(* CODESYS project 1210_xlh_terminal_manager.project
   Description: Receives some incoming messages and echoes them with CAN-ID +1
   Company: 3S - Smart Software Solutions GmbH
   Version: 1.0.0.0
   Title: CAN Bus API Example
   Author: 3S - Smart Software Solutions GmbH

Project tree, tasks and I/O mapping:
  xLH_base : CODESYS Control for Raspberry Pi 64 SL, CODESYS, order no. 2302000009, version 4.20.0.0
    application app
      libraries: Standard, 3.5.22.0 (System); Util, 3.5.22.0 (System); VisuDialogs, * (System); Memory, * (3S - Smart Software Solutions GmbH); CmpBitmapPool, * (System); CAN API, 1.0.0.4 (CODESYS); MemoryUtils, * (3S - Smart Software Solutions GmbH); CAA CiA 405, 4.3.0.0 (CODESYS)
      task CAN_OPEN_TASK (cyclic, interval 1 ms, priority 0) calls nothing
      task VISU_TASK (cyclic, interval 100 ms, priority 31) calls VisuElems.Visu_Prg
      task MAIN_TASK (cyclic, interval 4 ms, priority 1) calls MAIN_CALLER
      program MAIN_CALLER [ST]
      function block FB_SDO_READ_4_BYTE [ST]
      visualisation Visualization
      trace Trace (task MAIN_TASK): MAIN.diPosition, MAIN.iSetSpeed, MAIN.iDebug2Pos, MAIN.iDebug1Mileage, MAIN.auiUltrasonic[1], MAIN.fbReadStatusLoopTime.udiValue, MAIN.iSpeed2, MAIN.iSpeed1, MAIN.iPitch
      data type MOTION_CONTROL_BYTE
      program MAIN [ST]
      function block FB_XLH_TERMINAL [ST]: read, write
      TOOLBOX/
        GPIO/
          function block FB_XLH_GPIO [CFC]
          function block FB_XLH_SWITCH_BUTTON_LED [CFC]
        data type RGB
        data type UNION_BYTE_INT
      program io [ST]
    CANbus : CANbus, CODESYS, version 4.3.0.0
        settings: Baudrate = 1000 kbit/s
      CANopen_Manager : CANopen_Manager, CODESYS, version 4.3.0.0
          settings: NMT Start All = TRUE; Polling of optional slaves = FALSE; ConfigVersion = 50659584
        xlh_terminal : xlh_terminal, xemax ag, order no. 0, version Revision=16#00000001, FileVersion=1.0
            settings: NODEIDSAVED = 3; SDO Timeout = 1000000; PDO_Autoconfig = FALSE; EXPERTSETTINGS = FALSE; PDO 16#1400.COBID = 16#00000203; Process by CANopenManager = TRUE; PDO 16#1401.COBID = 16#00000303; Process by CANopenManager = TRUE; PDO 16#1402.COBID = 16#00000403; Process by CANopenManager = TRUE; PDO 16#1403.COBID = 16#00000503; Process by CANopenManager = TRUE; PDO 16#1800.COBID = 16#00000183; Process by CANopenManager = TRUE; PDO 16#1801.COBID = 16#00000283; Process by CANopenManager = TRUE; PDO 16#1802.COBID = 16#00000383; Process by CANopenManager = TRUE; PDO 16#1803.COBID = 16#00000483; Process by CANopenManager = TRUE; Data out 1 Byte 0.Subindex = 16#01; Data out 1 Byte 1.Subindex = 16#02; Data out 1 Byte 2.Subindex = 16#03; Data out 1 Byte 3.Subindex = 16#04; Data out 1 Byte 4.Subindex = 16#05; Data out 1 Byte 5.Subindex = 16#06; Data out 1 Byte 6.Subindex = 16#07; Data out 1 Byte 7.Subindex = 16#08; Data out 2 Byte 0.Subindex = 16#01; Data out 2 Byte 1.Subindex = 16#02; Data out 2 Byte 2.Subindex = 16#03; Data out 2 Byte 3.Subindex = 16#04; Data out 2 Byte 4.Subindex = 16#05; Data out 2 Byte 5.Subindex = 16#06; Data out 2 Byte 6.Subindex = 16#07; Data out 2 Byte 7.Subindex = 16#08; Data out 3 Byte 0.Subindex = 16#01; Data out 3 Byte 1.Subindex = 16#02; Data out 3 Byte 2.Subindex = 16#03; Data out 3 Byte 3.Subindex = 16#04;
              Data out 3 Byte 4.Subindex = 16#05; Data out 3 Byte 5.Subindex = 16#06; Data out 3 Byte 6.Subindex = 16#07; Data out 3 Byte 7.Subindex = 16#08; Data out 4 Byte 0.Subindex = 16#01; Data out 4 Byte 1.Subindex = 16#02; Data out 4 Byte 2.Subindex = 16#03; Data out 4 Byte 3.Subindex = 16#04; Data out 4 Byte 4.Subindex = 16#05; Data out 4 Byte 5.Subindex = 16#06; Data out 4 Byte 6.Subindex = 16#07; Data out 4 Byte 7.Subindex = 16#08; Data in 1 Byte 0.Subindex = 16#01; Data in 1 Byte 1.Subindex = 16#02; Data in 1 Byte 2.Subindex = 16#03; Data in 1 Byte 3.Subindex = 16#04; Data in 1 Byte 4.Subindex = 16#05; Data in 1 Byte 5.Subindex = 16#06; Data in 1 Byte 6.Subindex = 16#07; Data in 1 Byte 7.Subindex = 16#08; Data in 2 Byte 0.Subindex = 16#01; Data in 2 Byte 1.Subindex = 16#02; Data in 2 Byte 2.Subindex = 16#03; Data in 2 Byte 3.Subindex = 16#04; Data in 2 Byte 4.Subindex = 16#05; Data in 2 Byte 5.Subindex = 16#06; Data in 2 Byte 6.Subindex = 16#07; Data in 2 Byte 7.Subindex = 16#08; Data in 3 Byte 0.Subindex = 16#01; Data in 3 Byte 1.Subindex = 16#02; Data in 3 Byte 2.Subindex = 16#03; Data in 3 Byte 3.Subindex = 16#04; Data in 3 Byte 4.Subindex = 16#05; Data in 3 Byte 5.Subindex = 16#06; Data in 3 Byte 6.Subindex = 16#07; Data in 3 Byte 7.Subindex = 16#08; Data in 4 Byte 0.Subindex = 16#01; Data in 4 Byte 1.Subindex = 16#02; Data in 4 Byte 2.Subindex = 16#03; Data in 4 Byte 3.Subindex = 16#04;
              Data in 4 Byte 4.Subindex = 16#05; Data in 4 Byte 5.Subindex = 16#06; Data in 4 Byte 6.Subindex = 16#07; Data in 4 Byte 7.Subindex = 16#08; SDO List.Set COB-ID sync.Index = 16#1005; SDO List.Set COB-ID sync.Subindex = 16#00; SDO List.Set COB-ID sync.Value = 16#00000080; SDO List.Set COB-ID sync.Size = 32; SDO List.Set COB-ID sync.AbortIfError = FALSE; SDO List.Set COB-ID sync.JumpToLine = FALSE; SDO List.Set COB-ID sync.Line = 0; SDO List.Set communication cycle period.Index = 16#1006; SDO List.Set communication cycle period.Subindex = 16#00; SDO List.Set communication cycle period.Value = 16#00000000; SDO List.Set communication cycle period.Size = 32; SDO List.Set communication cycle period.AbortIfError = FALSE; SDO List.Set communication cycle period.JumpToLine = FALSE; SDO List.Set communication cycle period.Line = 0; SDO List.Set Guardtime.Index = 16#100C; SDO List.Set Guardtime.Subindex = 16#00; SDO List.Set Guardtime.Value = 16#000000C8; SDO List.Set Guardtime.Size = 16; SDO List.Set Guardtime.AbortIfError = FALSE; SDO List.Set Guardtime.JumpToLine = FALSE; SDO List.Set Guardtime.Line = 0; SDO List.Set Lifetime.Index = 16#100D; SDO List.Set Lifetime.Subindex = 16#00; SDO List.Set Lifetime.Value = 16#00000003; SDO List.Set Lifetime.Size = 8; SDO List.Set Lifetime.AbortIfError = FALSE; SDO List.Set Lifetime.JumpToLine = FALSE; SDO List.Set Lifetime.Line = 0; SDO List.Set Heartbeat Consumer.Index = 16#1016; SDO List.Set Heartbeat Consumer.Subindex = 16#01; SDO List.Set Heartbeat Consumer.Value = 0; SDO List.Set Heartbeat Consumer.Size = 32; SDO List.Set Heartbeat Consumer.AbortIfError = FALSE; SDO List.Set Heartbeat Consumer.JumpToLine = FALSE; SDO List.Set Heartbeat Consumer.Line = 0; SDO List.Disable PDO.Index = 16#1400;
              SDO List.Disable PDO.Subindex = 16#01; SDO List.Disable PDO.Value = 16#80000203; SDO List.Disable PDO.Size = 32; SDO List.Disable PDO.AbortIfError = FALSE; SDO List.Disable PDO.JumpToLine = FALSE; SDO List.Disable PDO.Line = 0; SDO List.Set transmission type.Index = 16#1400; SDO List.Set transmission type.Subindex = 16#02; SDO List.Set transmission type.Value = 16#FF; SDO List.Set transmission type.Size = 8; SDO List.Set transmission type.AbortIfError = FALSE; SDO List.Set transmission type.JumpToLine = FALSE; SDO List.Set transmission type.Line = 0; SDO List.Set and enable COB-ID.Index = 16#1400; SDO List.Set and enable COB-ID.Subindex = 16#01; SDO List.Set and enable COB-ID.Value = 16#00000203; SDO List.Set and enable COB-ID.Size = 32; SDO List.Set and enable COB-ID.AbortIfError = FALSE; SDO List.Set and enable COB-ID.JumpToLine = FALSE; SDO List.Set and enable COB-ID.Line = 0; SDO List.Disable PDO.Index = 16#1401; SDO List.Disable PDO.Subindex = 16#01; SDO List.Disable PDO.Value = 16#80000303; SDO List.Disable PDO.Size = 32; SDO List.Disable PDO.AbortIfError = FALSE; SDO List.Disable PDO.JumpToLine = FALSE; SDO List.Disable PDO.Line = 0; SDO List.Set transmission type.Index = 16#1401; SDO List.Set transmission type.Subindex = 16#02; SDO List.Set transmission type.Value = 16#FF; SDO List.Set transmission type.Size = 8; SDO List.Set transmission type.AbortIfError = FALSE; SDO List.Set transmission type.JumpToLine = FALSE; SDO List.Set transmission type.Line = 0; SDO List.Set and enable COB-ID.Index = 16#1401; SDO List.Set and enable COB-ID.Subindex = 16#01; SDO List.Set and enable COB-ID.Value = 16#00000303; SDO List.Set and enable COB-ID.Size = 32; SDO List.Set and enable COB-ID.AbortIfError = FALSE; SDO List.Set and enable COB-ID.JumpToLine = FALSE;
              SDO List.Set and enable COB-ID.Line = 0; SDO List.Disable PDO.Index = 16#1402; SDO List.Disable PDO.Subindex = 16#01; SDO List.Disable PDO.Value = 16#80000403; SDO List.Disable PDO.Size = 32; SDO List.Disable PDO.AbortIfError = FALSE; SDO List.Disable PDO.JumpToLine = FALSE; SDO List.Disable PDO.Line = 0; SDO List.Set transmission type.Index = 16#1402; SDO List.Set transmission type.Subindex = 16#02; SDO List.Set transmission type.Value = 16#FF; SDO List.Set transmission type.Size = 8; SDO List.Set transmission type.AbortIfError = FALSE; SDO List.Set transmission type.JumpToLine = FALSE; SDO List.Set transmission type.Line = 0; SDO List.Set and enable COB-ID.Index = 16#1402; SDO List.Set and enable COB-ID.Subindex = 16#01; SDO List.Set and enable COB-ID.Value = 16#00000403; SDO List.Set and enable COB-ID.Size = 32; SDO List.Set and enable COB-ID.AbortIfError = FALSE; SDO List.Set and enable COB-ID.JumpToLine = FALSE; SDO List.Set and enable COB-ID.Line = 0; SDO List.Disable PDO.Index = 16#1403; SDO List.Disable PDO.Subindex = 16#01; SDO List.Disable PDO.Value = 16#80000503; SDO List.Disable PDO.Size = 32; SDO List.Disable PDO.AbortIfError = FALSE; SDO List.Disable PDO.JumpToLine = FALSE; SDO List.Disable PDO.Line = 0; SDO List.Set transmission type.Index = 16#1403; SDO List.Set transmission type.Subindex = 16#02; SDO List.Set transmission type.Value = 16#FF; SDO List.Set transmission type.Size = 8; SDO List.Set transmission type.AbortIfError = FALSE; SDO List.Set transmission type.JumpToLine = FALSE; SDO List.Set transmission type.Line = 0; SDO List.Set and enable COB-ID.Index = 16#1403; SDO List.Set and enable COB-ID.Subindex = 16#01; SDO List.Set and enable COB-ID.Value = 16#00000503; SDO List.Set and enable COB-ID.Size = 32;
              SDO List.Set and enable COB-ID.AbortIfError = FALSE; SDO List.Set and enable COB-ID.JumpToLine = FALSE; SDO List.Set and enable COB-ID.Line = 0; SDO List.Disable PDO.Index = 16#1800; SDO List.Disable PDO.Subindex = 16#01; SDO List.Disable PDO.Value = 16#80000183; SDO List.Disable PDO.Size = 32; SDO List.Disable PDO.AbortIfError = FALSE; SDO List.Disable PDO.JumpToLine = FALSE; SDO List.Disable PDO.Line = 0; SDO List.Set transmission type.Index = 16#1800; SDO List.Set transmission type.Subindex = 16#02; SDO List.Set transmission type.Value = 16#FF; SDO List.Set transmission type.Size = 8; SDO List.Set transmission type.AbortIfError = FALSE; SDO List.Set transmission type.JumpToLine = FALSE; SDO List.Set transmission type.Line = 0; SDO List.Set inhibit time.Index = 16#1800; SDO List.Set inhibit time.Subindex = 16#03; SDO List.Set inhibit time.Value = 16#0000; SDO List.Set inhibit time.Size = 16; SDO List.Set inhibit time.AbortIfError = FALSE; SDO List.Set inhibit time.JumpToLine = FALSE; SDO List.Set inhibit time.Line = 0; SDO List.Set event time.Index = 16#1800; SDO List.Set event time.Subindex = 16#05; SDO List.Set event time.Value = 16#0000; SDO List.Set event time.Size = 16; SDO List.Set event time.AbortIfError = FALSE; SDO List.Set event time.JumpToLine = FALSE; SDO List.Set event time.Line = 0; SDO List.Set and enable COB-ID.Index = 16#1800; SDO List.Set and enable COB-ID.Subindex = 16#01; SDO List.Set and enable COB-ID.Value = 16#00000183; SDO List.Set and enable COB-ID.Size = 32; SDO List.Set and enable COB-ID.AbortIfError = FALSE; SDO List.Set and enable COB-ID.JumpToLine = FALSE; SDO List.Set and enable COB-ID.Line = 0; SDO List.Disable PDO.Index = 16#1801; SDO List.Disable PDO.Subindex = 16#01;
              SDO List.Disable PDO.Value = 16#80000283; SDO List.Disable PDO.Size = 32; SDO List.Disable PDO.AbortIfError = FALSE; SDO List.Disable PDO.JumpToLine = FALSE; SDO List.Disable PDO.Line = 0; SDO List.Set transmission type.Index = 16#1801; SDO List.Set transmission type.Subindex = 16#02; SDO List.Set transmission type.Value = 16#FF; SDO List.Set transmission type.Size = 8; SDO List.Set transmission type.AbortIfError = FALSE; SDO List.Set transmission type.JumpToLine = FALSE; SDO List.Set transmission type.Line = 0; SDO List.Set inhibit time.Index = 16#1801; SDO List.Set inhibit time.Subindex = 16#03; SDO List.Set inhibit time.Value = 16#0000; SDO List.Set inhibit time.Size = 16; SDO List.Set inhibit time.AbortIfError = FALSE; SDO List.Set inhibit time.JumpToLine = FALSE; SDO List.Set inhibit time.Line = 0; SDO List.Set event time.Index = 16#1801; SDO List.Set event time.Subindex = 16#05; SDO List.Set event time.Value = 16#0000; SDO List.Set event time.Size = 16; SDO List.Set event time.AbortIfError = FALSE; SDO List.Set event time.JumpToLine = FALSE; SDO List.Set event time.Line = 0; SDO List.Set and enable COB-ID.Index = 16#1801; SDO List.Set and enable COB-ID.Subindex = 16#01; SDO List.Set and enable COB-ID.Value = 16#00000283; SDO List.Set and enable COB-ID.Size = 32; SDO List.Set and enable COB-ID.AbortIfError = FALSE; SDO List.Set and enable COB-ID.JumpToLine = FALSE; SDO List.Set and enable COB-ID.Line = 0; SDO List.Disable PDO.Index = 16#1802; SDO List.Disable PDO.Subindex = 16#01; SDO List.Disable PDO.Value = 16#80000383; SDO List.Disable PDO.Size = 32; SDO List.Disable PDO.AbortIfError = FALSE; SDO List.Disable PDO.JumpToLine = FALSE; SDO List.Disable PDO.Line = 0;
              SDO List.Set transmission type.Index = 16#1802; SDO List.Set transmission type.Subindex = 16#02; SDO List.Set transmission type.Value = 16#FF; SDO List.Set transmission type.Size = 8; SDO List.Set transmission type.AbortIfError = FALSE; SDO List.Set transmission type.JumpToLine = FALSE; SDO List.Set transmission type.Line = 0; SDO List.Set inhibit time.Index = 16#1802; SDO List.Set inhibit time.Subindex = 16#03; SDO List.Set inhibit time.Value = 16#0000; SDO List.Set inhibit time.Size = 16; SDO List.Set inhibit time.AbortIfError = FALSE; SDO List.Set inhibit time.JumpToLine = FALSE; SDO List.Set inhibit time.Line = 0; SDO List.Set event time.Index = 16#1802; SDO List.Set event time.Subindex = 16#05; SDO List.Set event time.Value = 16#0000; SDO List.Set event time.Size = 16; SDO List.Set event time.AbortIfError = FALSE; SDO List.Set event time.JumpToLine = FALSE; SDO List.Set event time.Line = 0; SDO List.Set and enable COB-ID.Index = 16#1802; SDO List.Set and enable COB-ID.Subindex = 16#01; SDO List.Set and enable COB-ID.Value = 16#00000383; SDO List.Set and enable COB-ID.Size = 32; SDO List.Set and enable COB-ID.AbortIfError = FALSE; SDO List.Set and enable COB-ID.JumpToLine = FALSE; SDO List.Set and enable COB-ID.Line = 0; SDO List.Disable PDO.Index = 16#1803; SDO List.Disable PDO.Subindex = 16#01; SDO List.Disable PDO.Value = 16#80000483; SDO List.Disable PDO.Size = 32; SDO List.Disable PDO.AbortIfError = FALSE; SDO List.Disable PDO.JumpToLine = FALSE; SDO List.Disable PDO.Line = 0; SDO List.Set transmission type.Index = 16#1803; SDO List.Set transmission type.Subindex = 16#02; SDO List.Set transmission type.Value = 16#FF; SDO List.Set transmission type.Size = 8; SDO List.Set transmission type.AbortIfError = FALSE;
              SDO List.Set transmission type.JumpToLine = FALSE; SDO List.Set transmission type.Line = 0; SDO List.Set inhibit time.Index = 16#1803; SDO List.Set inhibit time.Subindex = 16#03; SDO List.Set inhibit time.Value = 16#0000; SDO List.Set inhibit time.Size = 16; SDO List.Set inhibit time.AbortIfError = FALSE; SDO List.Set inhibit time.JumpToLine = FALSE; SDO List.Set inhibit time.Line = 0; SDO List.Set event time.Index = 16#1803; SDO List.Set event time.Subindex = 16#05; SDO List.Set event time.Value = 16#0000; SDO List.Set event time.Size = 16; SDO List.Set event time.AbortIfError = FALSE; SDO List.Set event time.JumpToLine = FALSE; SDO List.Set event time.Line = 0; SDO List.Set and enable COB-ID.Index = 16#1803; SDO List.Set and enable COB-ID.Subindex = 16#01; SDO List.Set and enable COB-ID.Value = 16#00000483; SDO List.Set and enable COB-ID.Size = 32; SDO List.Set and enable COB-ID.AbortIfError = FALSE; SDO List.Set and enable COB-ID.JumpToLine = FALSE; SDO List.Set and enable COB-ID.Line = 0; ConfigVersion = 50659584
            output app.MAIN.fbTerminal.abyOutData1[0] : USINT  // Data out 1 Byte 0
            output app.MAIN.fbTerminal.abyOutData1[1] : USINT  // Data out 1 Byte 1
            output app.MAIN.fbTerminal.abyOutData1[2] : USINT  // Data out 1 Byte 2
            output app.MAIN.fbTerminal.abyOutData1[3] : USINT  // Data out 1 Byte 3
            output app.MAIN.fbTerminal.abyOutData1[4] : USINT  // Data out 1 Byte 4
            output app.MAIN.fbTerminal.abyOutData1[5] : USINT  // Data out 1 Byte 5
            output app.MAIN.fbTerminal.abyOutData1[6] : USINT  // Data out 1 Byte 6
            output app.MAIN.fbTerminal.abyOutData1[7] : USINT  // Data out 1 Byte 7
            output app.MAIN.fbTerminal.abyOutData2[0] : USINT  // Data out 2 Byte 0
            output app.MAIN.fbTerminal.abyOutData2[1] : USINT  // Data out 2 Byte 1
            output app.MAIN.fbTerminal.abyOutData2[2] : USINT  // Data out 2 Byte 2
            output app.MAIN.fbTerminal.abyOutData2[3] : USINT  // Data out 2 Byte 3
            output app.MAIN.fbTerminal.abyOutData2[4] : USINT  // Data out 2 Byte 4
            output app.MAIN.fbTerminal.abyOutData2[5] : USINT  // Data out 2 Byte 5
            output app.MAIN.fbTerminal.abyOutData2[6] : USINT  // Data out 2 Byte 6
            output app.MAIN.fbTerminal.abyOutData2[7] : USINT  // Data out 2 Byte 7
            output app.MAIN.fbTerminal.abyOutData3[0] : USINT  // Data out 3 Byte 0
            output app.MAIN.fbTerminal.abyOutData3[1] : USINT  // Data out 3 Byte 1
            output app.MAIN.fbTerminal.abyOutData3[2] : USINT  // Data out 3 Byte 2
            output app.MAIN.fbTerminal.abyOutData3[3] : USINT  // Data out 3 Byte 3
            output app.MAIN.fbTerminal.abyOutData3[4] : USINT  // Data out 3 Byte 4
            output app.MAIN.fbTerminal.abyOutData3[5] : USINT  // Data out 3 Byte 5
            output app.MAIN.fbTerminal.abyOutData3[6] : USINT  // Data out 3 Byte 6
            output app.MAIN.fbTerminal.abyOutData3[7] : USINT  // Data out 3 Byte 7
            output app.MAIN.fbTerminal.abyOutData4[0] : USINT  // Data out 4 Byte 0
            output app.MAIN.fbTerminal.abyOutData4[1] : USINT  // Data out 4 Byte 1
            output app.MAIN.fbTerminal.abyOutData4[2] : USINT  // Data out 4 Byte 2
            output app.MAIN.fbTerminal.abyOutData4[3] : USINT  // Data out 4 Byte 3
            output app.MAIN.fbTerminal.abyOutData4[4] : USINT  // Data out 4 Byte 4
            output app.MAIN.fbTerminal.abyOutData4[5] : USINT  // Data out 4 Byte 5
            output app.MAIN.fbTerminal.abyOutData4[6] : USINT  // Data out 4 Byte 6
            output app.MAIN.fbTerminal.abyOutData4[7] : USINT  // Data out 4 Byte 7
            input  app.MAIN.fbTerminal.abyInData1[0] : USINT  // Data in 1 Byte 0
            input  app.MAIN.fbTerminal.abyInData1[1] : USINT  // Data in 1 Byte 1
            input  app.MAIN.fbTerminal.abyInData1[2] : USINT  // Data in 1 Byte 2
            input  app.MAIN.fbTerminal.abyInData1[3] : USINT  // Data in 1 Byte 3
            input  app.MAIN.fbTerminal.abyInData1[4] : USINT  // Data in 1 Byte 4
            input  app.MAIN.fbTerminal.abyInData1[5] : USINT  // Data in 1 Byte 5
            input  app.MAIN.fbTerminal.abyInData1[6] : USINT  // Data in 1 Byte 6
            input  app.MAIN.fbTerminal.abyInData1[7] : USINT  // Data in 1 Byte 7
            input  app.MAIN.fbTerminal.abyInData2[0] : USINT  // Data in 2 Byte 0
            input  app.MAIN.fbTerminal.abyInData2[1] : USINT  // Data in 2 Byte 1
            input  app.MAIN.fbTerminal.abyInData2[2] : USINT  // Data in 2 Byte 2
            input  app.MAIN.fbTerminal.abyInData2[3] : USINT  // Data in 2 Byte 3
            input  app.MAIN.fbTerminal.abyInData2[4] : USINT  // Data in 2 Byte 4
            input  app.MAIN.fbTerminal.abyInData2[5] : USINT  // Data in 2 Byte 5
            input  app.MAIN.fbTerminal.abyInData2[6] : USINT  // Data in 2 Byte 6
            input  app.MAIN.fbTerminal.abyInData2[7] : USINT  // Data in 2 Byte 7
            input  app.MAIN.fbTerminal.abyInData3[0] : USINT  // Data in 3 Byte 0
            input  app.MAIN.fbTerminal.abyInData3[1] : USINT  // Data in 3 Byte 1
            input  app.MAIN.fbTerminal.abyInData3[2] : USINT  // Data in 3 Byte 2
            input  app.MAIN.fbTerminal.abyInData3[3] : USINT  // Data in 3 Byte 3
            input  app.MAIN.fbTerminal.abyInData3[4] : USINT  // Data in 3 Byte 4
            input  app.MAIN.fbTerminal.abyInData3[5] : USINT  // Data in 3 Byte 5
            input  app.MAIN.fbTerminal.abyInData3[6] : USINT  // Data in 3 Byte 6
            input  app.MAIN.fbTerminal.abyInData3[7] : USINT  // Data in 3 Byte 7
            input  app.MAIN.fbTerminal.abyInData4[0] : USINT  // Data in 4 Byte 0
            input  app.MAIN.fbTerminal.abyInData4[1] : USINT  // Data in 4 Byte 1
            input  app.MAIN.fbTerminal.abyInData4[2] : USINT  // Data in 4 Byte 2
            input  app.MAIN.fbTerminal.abyInData4[3] : USINT  // Data in 4 Byte 3
            input  app.MAIN.fbTerminal.abyInData4[4] : USINT  // Data in 4 Byte 4
            input  app.MAIN.fbTerminal.abyInData4[5] : USINT  // Data in 4 Byte 5
            input  app.MAIN.fbTerminal.abyInData4[6] : USINT  // Data in 4 Byte 6
            input  app.MAIN.fbTerminal.abyInData4[7] : USINT  // Data in 4 Byte 7
    Camera device
      <Leer>
    GPIOs_A_B : GPIOs B+/Pi2, CODESYS, version 4.20.0.0
        input  app.io.gpio.bSw1 : BOOL  // digital inputs (GPIO0..GPIO31).Bit4
        input  app.io.gpio.bSw2 : BOOL  // digital inputs (GPIO0..GPIO31).Bit5
        input  app.io.gpio.bSw3 : BOOL  // digital inputs (GPIO0..GPIO31).Bit6
        input  app.io.gpio.bSw4 : BOOL  // digital inputs (GPIO0..GPIO31).Bit12
        input  app.io.gpio.bSw5 : BOOL  // digital inputs (GPIO0..GPIO31).Bit13
        input  app.io.gpio.bSw6 : BOOL  // digital inputs (GPIO0..GPIO31).Bit16
        input  app.io.gpio.bSw7 : BOOL  // digital inputs (GPIO0..GPIO31).Bit17
        input  app.io.gpio.bSw8 : BOOL  // digital inputs (GPIO0..GPIO31).Bit19
        output app.io.gpio.bLed1 : BOOL  // digital outputs (GPIO0..GPIO31).Bit20
        output app.io.gpio.bLed2 : BOOL  // digital outputs (GPIO0..GPIO31).Bit21
        output app.io.gpio.bLed3 : BOOL  // digital outputs (GPIO0..GPIO31).Bit22
        output app.io.gpio.bLed4 : BOOL  // digital outputs (GPIO0..GPIO31).Bit23
        output app.io.gpio.bLed5 : BOOL  // digital outputs (GPIO0..GPIO31).Bit24
        output app.io.gpio.bLed6 : BOOL  // digital outputs (GPIO0..GPIO31).Bit26
        output app.io.gpio.bLed7 : BOOL  // digital outputs (GPIO0..GPIO31).Bit27
        unmapped channels: digital inputs (GPIO0..GPIO31), digital outputs (GPIO0..GPIO31)
    I²C
    SoftMotion General Axis Pool
      x_axis : SM_Drive_PosControl, CODESYS, order no. 1805, version 4.18.0.0
          settings: dwRatioTechUnitsDenom = 101846; iRatioTechUnitsNum = 125; eRampType = 1; fSWMaxVelocity = 50; fSWMaxAcceleration = 100; fSWMaxDeceleration = 100; fSWMaxJerk = 1000; fSWLimitNegative = -1000; ScalingIncs = 814768; ScalingUnits = 1000; IsLinearMotor = TRUE; MaximumOutputVelocityInt = 40738; MinimumOutputVelocityInt = -40738; Kp = 0.05; MaxFollowingError = 5.0; EnableFollowingErrorCheck = TRUE; DeadTime = 3.0
      z_axis : SM_Drive_PosControl, CODESYS, order no. 1805, version 4.18.0.0
          settings: wDriveID = 3; dwRatioTechUnitsDenom = 101846; iRatioTechUnitsNum = 125; eRampType = 1; fSWMaxVelocity = 50; fSWMaxAcceleration = 100; fSWMaxDeceleration = 100; fSWMaxJerk = 1000; fSWLimitNegative = -1000; ScalingIncs = 814768; ScalingUnits = 1000; IsLinearMotor = TRUE; MaximumOutputVelocityInt = 40738; MinimumOutputVelocityInt = -40738; Kp = 0.05; MaxFollowingError = 5.0; EnableFollowingErrorCheck = TRUE; DeadTime = 3.0
      y_axis : SM_Drive_PosControl, CODESYS, order no. 1805, version 4.18.0.0
          settings: wDriveID = 2; dwRatioTechUnitsDenom = 101846; iRatioTechUnitsNum = 125; eRampType = 1; fSWMaxVelocity = 50; fSWMaxAcceleration = 100; fSWMaxDeceleration = 100; fSWMaxJerk = 1000; fSWLimitNegative = -1000; ScalingIncs = 814768; ScalingUnits = 1000; IsLinearMotor = TRUE; MaximumOutputVelocityInt = 40738; MinimumOutputVelocityInt = -40738; Kp = 0.05; MaxFollowingError = 5.0; EnableFollowingErrorCheck = TRUE; DeadTime = 3.0
      a_axis : SM_Drive_PosControl, CODESYS, order no. 1805, version 4.18.0.0
          settings: wDriveID = 4; dwRatioTechUnitsDenom = 101846; iRatioTechUnitsNum = -125; eRampType = 1; fSWMaxVelocity = 50; fSWMaxAcceleration = 100; fSWMaxDeceleration = 100; fSWMaxJerk = 1000; fSWLimitNegative = -1000.0; ScalingIncs = 814768; ScalingUnits = 1000; InvertDirection = TRUE; IsLinearMotor = TRUE; MaximumOutputVelocityInt = 40738; MinimumOutputVelocityInt = -40738; Kp = 0.05; MaxFollowingError = 5.0; EnableFollowingErrorCheck = TRUE; DeadTime = 3.0
    Onewire
    SPI
  libraries: VisuSymbols, 4.5.0.0 (System); DepictorBase, 1.2.0.0 (CODESYS)
  text list GlobalTextList
  5ce3da45-db07-42e7-a21c-a00fff4ed8f6|C:\Users\phe\Downloads\Musterloesung_FUP.PNG
*)

// xLH_base/app/MOTION_CONTROL_BYTE
TYPE MOTION_CONTROL_BYTE :
STRUCT
	bEnable: BOOL;
	bDir: BOOL;
	bReset: BOOL;
	bInverted: BOOL;
	bInMotion: BOOL;
	bMoveWithoutPulse: BOOL;
END_STRUCT
END_TYPE

// xLH_base/app/TOOLBOX/RGB
{attribute 'qualified_only'}
{attribute 'strict'}
TYPE RGB :
(
	OFF := 0,
	RED := 1,
	GREEN := 2,
	BLUE := 3
);
END_TYPE

// xLH_base/app/TOOLBOX/UNION_BYTE_INT
TYPE UNION_BYTE_INT :
UNION
	uiInt: UINT;;
	iInt: INT;
	abyStream: ARRAY[0..1] OF BYTE;	
END_UNION
END_TYPE

// xLH_base/app/MAIN_CALLER
PROGRAM MAIN_CALLER
VAR
	bDevicesCoRunning: BOOL;
	fbTonDevicesCoRunning: TON := (PT:=T#250MS);
END_VAR

// Ueberwachung ob alle CAN-Open Devices im Status RUN sind
fbTonDevicesCoRunning(IN:= xlh_terminal.CANopenState = _3SCOS.DEVICE_STATE.OPERATIONAL);

// falls alle Devices im Status RUN sind (inklusive Verzögerung), wird die POE MAIN aufgerufen
IF fbTonDevicesCoRunning.Q THEN
	MAIN();
END_IF

END_PROGRAM

// xLH_base/app/MAIN
PROGRAM MAIN
VAR
	byDummy: BYTE;
	udiDummy: UDINT;
	
	fbTerminal: FB_XLH_TERMINAL;
	
	fbBlink: BLINK := (TIMEHIGH:=T#100MS, TIMELOW:=T#100MS, ENABLE:=TRUE);
	fbReadStatusRefreshTime: FB_SDO_READ_4_BYTE;
	fbReadStatusLoopTime: FB_SDO_READ_4_BYTE;
	bStartup: BOOL := TRUE;
END_VAR

IF bStartup THEN
	bStartup := FALSE;
END_IF

fbTerminal.read();

(*
fbTerminal.abyOutData1[0] := fbTerminal.abyOutData1[0] + 1;
fbTerminal.abyOutData2[0] := fbTerminal.abyOutData2[0] + 1;
fbTerminal.abyOutData3[0] := fbTerminal.abyOutData3[0] + 1;
fbTerminal.abyOutData4[0] := fbTerminal.abyOutData4[0] + 1;
*)

io.gpio.bLed1 := (fbTerminal.abyInData1[0] <> 0);
io.gpio.bLed2 := (fbTerminal.abyInData2[0] <> 0);


byDummy := fbTerminal.abyInData1[0];
byDummy := fbTerminal.abyInData1[1];
byDummy := fbTerminal.abyInData1[2];
byDummy := fbTerminal.abyInData1[3];
byDummy := fbTerminal.abyInData1[4];
byDummy := fbTerminal.abyInData1[5];
byDummy := fbTerminal.abyInData1[6];
byDummy := fbTerminal.abyInData1[7];

byDummy := fbTerminal.abyInData2[0];
byDummy := fbTerminal.abyInData2[1];
byDummy := fbTerminal.abyInData2[2];
byDummy := fbTerminal.abyInData2[3];
byDummy := fbTerminal.abyInData2[4];
byDummy := fbTerminal.abyInData2[5];
byDummy := fbTerminal.abyInData2[6];
byDummy := fbTerminal.abyInData2[7];

byDummy := fbTerminal.abyInData3[0];
byDummy := fbTerminal.abyInData3[1];
byDummy := fbTerminal.abyInData3[2];
byDummy := fbTerminal.abyInData3[3];
byDummy := fbTerminal.abyInData3[4];
byDummy := fbTerminal.abyInData3[5];
byDummy := fbTerminal.abyInData3[6];
byDummy := fbTerminal.abyInData3[7];

byDummy := fbTerminal.abyInData4[0];
byDummy := fbTerminal.abyInData4[1];
byDummy := fbTerminal.abyInData4[2];
byDummy := fbTerminal.abyInData4[3];
byDummy := fbTerminal.abyInData4[4];
byDummy := fbTerminal.abyInData4[5];
byDummy := fbTerminal.abyInData4[6];
byDummy := fbTerminal.abyInData4[7];

byDummy := fbTerminal.abyOutData1[0];
byDummy := fbTerminal.abyOutData1[1];
byDummy := fbTerminal.abyOutData1[2];
byDummy := fbTerminal.abyOutData1[3];
byDummy := fbTerminal.abyOutData1[4];
byDummy := fbTerminal.abyOutData1[5];
byDummy := fbTerminal.abyOutData1[6];
byDummy := fbTerminal.abyOutData1[7];

byDummy := fbTerminal.abyOutData2[0];
byDummy := fbTerminal.abyOutData2[1];
byDummy := fbTerminal.abyOutData2[2];
byDummy := fbTerminal.abyOutData2[3];
byDummy := fbTerminal.abyOutData2[4];
byDummy := fbTerminal.abyOutData2[5];
byDummy := fbTerminal.abyOutData2[6];
byDummy := fbTerminal.abyOutData2[7];

byDummy := fbTerminal.abyOutData3[0];
byDummy := fbTerminal.abyOutData3[1];
byDummy := fbTerminal.abyOutData3[2];
byDummy := fbTerminal.abyOutData3[3];
byDummy := fbTerminal.abyOutData3[4];
byDummy := fbTerminal.abyOutData3[5];
byDummy := fbTerminal.abyOutData3[6];
byDummy := fbTerminal.abyOutData3[7];

byDummy := fbTerminal.abyOutData4[0];
byDummy := fbTerminal.abyOutData4[1];
byDummy := fbTerminal.abyOutData4[2];
byDummy := fbTerminal.abyOutData4[3];
byDummy := fbTerminal.abyOutData4[4];
byDummy := fbTerminal.abyOutData4[5];
byDummy := fbTerminal.abyOutData4[6];
byDummy := fbTerminal.abyOutData4[7];

fbTerminal.write();

// ##############################################################
(*
fbBlink();
fbReadStatusRefreshTime(
	bEnable:=fbBlink.OUT,
	usCoDeviceId:=xlh_terminal.NodeID,
	uiIndex:=16#5800, usSubindex:=1);
fbReadStatusLoopTime(
	bEnable:= NOT fbBlink.OUT,
	usCoDeviceId:=xlh_terminal.NodeID,
	uiIndex:=16#5800, usSubindex:=2);
udiDummy := fbReadStatusRefreshTime.udiValue;
udiDummy := fbReadStatusLoopTime.udiValue;
*)
// ##############################################################

END_PROGRAM

// xLH_base/app/io
PROGRAM io 
VAR_INPUT
	gpio: FB_XLH_GPIO;	
	sw_btn_led: FB_XLH_SWITCH_BUTTON_LED;	
END_VAR
VAR	

END_VAR

// Dynamixel ToDo
(*
Es Drehscheibe  7
Es Bahn Links   5
Es Bahn rechts  6
*)

END_PROGRAM

// xLH_base/app/TOOLBOX/GPIO/FB_XLH_GPIO
FUNCTION_BLOCK FB_XLH_GPIO
VAR_INPUT
	bLed1: BOOL;
	bLed2: BOOL;
	bLed3: BOOL;
	bLed4: BOOL;
	bLed5: BOOL;
	bLed6: BOOL;
	bLed7: BOOL;	
END_VAR
VAR_OUTPUT
	bSw1: BOOL;
	bSw2: BOOL;
	bSw3: BOOL;
	bSw4: BOOL;
	bSw5: BOOL;
	bSw6: BOOL;
	bSw7: BOOL;
	bSw8: BOOL;
END_VAR

END_FUNCTION_BLOCK

// xLH_base/app/TOOLBOX/GPIO/FB_XLH_SWITCH_BUTTON_LED
FUNCTION_BLOCK FB_XLH_SWITCH_BUTTON_LED
VAR_INPUT
	bLedSw0: BOOL;
	bLedSw1: BOOL;
	bLedSw2: BOOL;
	bLedSw3: BOOL;
	bLedSw4: BOOL;
	bLedSw5: BOOL;
	bLedSw6: BOOL;
	bLedSw7: BOOL;	
	bLedBtn0: BOOL;
	bLedBtn1: BOOL;
	bLedBtn2: BOOL;
	bLedBtn3: BOOL;
	bLedBtn4: BOOL;
	bLedBtn5: BOOL;
	bLedBtn6: BOOL;
	bLedBtn7: BOOL;	
END_VAR
VAR_OUTPUT
	bSw1: BOOL;
	bSw2: BOOL;
	bSw3: BOOL;
	bSw4: BOOL;
	bSw5: BOOL;
	bSw6: BOOL;
	bSw7: BOOL;
	bSw8: BOOL;
	bBtn1: BOOL;
	bBtn2: BOOL;
	bBtn3: BOOL;
	bBtn4: BOOL;
	bBtn5: BOOL;
	bBtn6: BOOL;
	bBtn7: BOOL;
	bBtn8: BOOL;
END_VAR

END_FUNCTION_BLOCK

// xLH_base/app/FB_XLH_TERMINAL
// =====================================================================
// FB_XLH_GPIO
// Pure data container for the GPIO control elements of the xLH board:
// 7 LEDs as inputs (written by the PLC program) and 8 switches as
// outputs (read from the board). The fields are mapped to the hardware
// via the device I/O configuration (CANopen); the read/write methods
// are currently empty and serve as extension hooks.
// =====================================================================
FUNCTION_BLOCK FB_XLH_TERMINAL
VAR_INPUT
	eRgbModeOff: RGB;
	eRgbModeManual: RGB;
	eRgbModeF1: RGB;
	eRgbModeF2: RGB;
	
	eRgbModeF3: RGB;
	eRgbAxXp: RGB;
	eRgbAxXm: RGB;
	eRgbAxYp: RGB;
	
	eRgbAxYm: RGB;
	eRgbAxZp: RGB;
	eRgbAxZm: RGB;
	eRgbAxCp: RGB;
	
	eRgbAxCm: RGB;
	eRgbMagnet: RGB;
	eRgbAxIncC: RGB;
	eRgbAxIncXY: RGB;
	
	eRgbAxIncZ: RGB;	
	eRgbVelMaster: RGB;	
	
	usBrightness: USINT := 50;
	
	{attribute 'displaymode':='hex'} 
	abyOutData1: ARRAY[0..7] OF BYTE;
	{attribute 'displaymode':='hex'}
	abyOutData2: ARRAY[0..7] OF BYTE;
	{attribute 'displaymode':='hex'}
	abyOutData3: ARRAY[0..7] OF BYTE;
	{attribute 'displaymode':='hex'}
	abyOutData4: ARRAY[0..7] OF BYTE;
END_VAR
VAR_OUTPUT
	bModeOff: BOOL;
	bModeManual: BOOL;
	bModeF1: BOOL;
	bModeF2: BOOL;
	bModeF3: BOOL;
	
	bAxXp: BOOL;
	bAxXm: BOOL;
	bAxYp: BOOL;
	bAxYm: BOOL;
	bAxZp: BOOL;
	bAxZm: BOOL;
	bAxCp: BOOL;
	bAxCm: BOOL;
	
	bMagnet: BOOL;
	
	iAxIncC: INT;
	bAxIncC: BOOL;
	iAxIncXY: INT;
	bAxIncXY: BOOL;
	iAxIncZ: INT;
	bAxIncZ: BOOL;
		
	iVelMaster: INT;	


	{attribute 'displaymode':='hex'} 
	abyInData1: ARRAY[0..7] OF BYTE;
	{attribute 'displaymode':='hex'}
	abyInData2: ARRAY[0..7] OF BYTE;
	{attribute 'displaymode':='hex'}
	abyInData3: ARRAY[0..7] OF BYTE;
	{attribute 'displaymode':='hex'}
	abyInData4: ARRAY[0..7] OF BYTE;
END_VAR

METHOD read : BOOL
VAR_INPUT
END_VAR
VAR
	unpackByte: MEM.UnpackByte;	
	value: UNION_BYTE_INT;
END_VAR
// PDO 1
unpackByte(byValue := abyInData1[0]);	
bModeOff := unpackByte.xBit0;
bAxIncC := unpackByte.xBit1;
bAxIncXY := unpackByte.xBit2;
bAxIncZ := unpackByte.xBit3;
bModeManual := unpackByte.xBit4;
bModeF1 := unpackByte.xBit5;
bAxCp := unpackByte.xBit6;
bAxYp := unpackByte.xBit7;

value.abyStream[0] := abyInData1[2];
value.abyStream[1] := abyInData1[3];
iAxIncC := value.iInt;

value.abyStream[0] := abyInData1[4];
value.abyStream[1] := abyInData1[5];
iAxIncXY := value.iInt;

value.abyStream[0] := abyInData1[6];
value.abyStream[1] := abyInData1[7];
iAxIncZ := value.iInt;


// PDO 2
unpackByte(byValue := abyInData2[0]);	
bAxZp := unpackByte.xBit0;
bModeF2 := unpackByte.xBit1;
bAxXm := unpackByte.xBit2;
bMagnet := unpackByte.xBit3;
bAxXp := unpackByte.xBit4;
bModeF3 := unpackByte.xBit5;
bAxCm := unpackByte.xBit6;
bAxYm := unpackByte.xBit7;

unpackByte(byValue := abyInData2[1]);	
bAxZm := unpackByte.xBit0;

value.abyStream[0] := abyInData2[2];
value.abyStream[1] := abyInData2[3];
iVelMaster := value.iInt;
END_METHOD

METHOD write : BOOL
VAR_INPUT
END_VAR
abyOutData1[0] := MEM.PackBitsToByte(
	((eRgbAxIncZ = RGB.GREEN) OR (eRgbAxIncZ = RGB.BLUE)),
	((eRgbAxIncZ = RGB.RED) OR (eRgbAxIncZ = RGB.BLUE)),
	//
	((eRgbAxIncXY = RGB.GREEN) OR (eRgbAxIncXY = RGB.BLUE)),
	((eRgbAxIncXY = RGB.RED) OR (eRgbAxIncXY = RGB.BLUE)),
	//
	((eRgbAxIncC = RGB.GREEN) OR (eRgbAxIncC = RGB.BLUE)),
	((eRgbAxIncC = RGB.RED) OR (eRgbAxIncC = RGB.BLUE)),
	//
	((eRgbModeOff = RGB.GREEN) OR (eRgbModeOff = RGB.BLUE)),
	((eRgbModeOff = RGB.RED) OR (eRgbModeOff = RGB.BLUE)));
	
	
abyOutData1[1] := MEM.PackBitsToByte(
	((eRgbAxYp = RGB.GREEN) OR (eRgbAxYp = RGB.BLUE)),
	((eRgbAxYp = RGB.RED) OR (eRgbAxYp = RGB.BLUE)),
	//
	((eRgbAxCp = RGB.GREEN) OR (eRgbAxCp = RGB.BLUE)),
	((eRgbAxCp = RGB.RED) OR (eRgbAxCp = RGB.BLUE)),
	//
	((eRgbModeF1 = RGB.GREEN) OR (eRgbModeF1 = RGB.BLUE)),
	((eRgbModeF1 = RGB.RED) OR (eRgbModeF1 = RGB.BLUE)),
	//
	((eRgbModeManual = RGB.GREEN) OR (eRgbModeManual = RGB.BLUE)),
	((eRgbModeManual = RGB.RED) OR (eRgbModeManual = RGB.BLUE)));
	

abyOutData1[2] := MEM.PackBitsToByte(
	((eRgbAxXm = RGB.GREEN) OR (eRgbAxXm = RGB.BLUE)),
	((eRgbAxXm = RGB.RED) OR (eRgbAxXm = RGB.BLUE)),
	//
	((eRgbVelMaster = RGB.GREEN) OR (eRgbVelMaster = RGB.BLUE)),
	((eRgbVelMaster = RGB.RED) OR (eRgbVelMaster = RGB.BLUE)),
	//
	((eRgbModeF2 = RGB.GREEN) OR (eRgbModeF2 = RGB.BLUE)),
	((eRgbModeF2 = RGB.RED) OR (eRgbModeF2 = RGB.BLUE)),
	//
	((eRgbAxZp = RGB.GREEN) OR (eRgbAxZp = RGB.BLUE)),
	((eRgbAxZp = RGB.RED) OR (eRgbAxZp = RGB.BLUE)));
	
	
abyOutData1[3] := MEM.PackBitsToByte(
	((eRgbAxCm = RGB.GREEN) OR (eRgbAxCm = RGB.BLUE)),
	((eRgbAxCm = RGB.RED) OR (eRgbAxCm = RGB.BLUE)),
	//
	((eRgbModeF3 = RGB.GREEN) OR (eRgbModeF3 = RGB.BLUE)),
	((eRgbModeF3 = RGB.RED) OR (eRgbModeF3 = RGB.BLUE)),
	//
	((eRgbAxXp = RGB.GREEN) OR (eRgbAxXp = RGB.BLUE)),
	((eRgbAxXp = RGB.RED) OR (eRgbAxXp = RGB.BLUE)),
	//
	((eRgbMagnet = RGB.GREEN) OR (eRgbMagnet = RGB.BLUE)),
	((eRgbMagnet = RGB.RED) OR (eRgbMagnet = RGB.BLUE)));
	

abyOutData1[4] := MEM.PackBitsToByte(
	FALSE,
	FALSE,
	FALSE,
	FALSE,
	//
	((eRgbAxZm = RGB.GREEN) OR (eRgbAxZm = RGB.BLUE)),
	((eRgbAxZm = RGB.RED) OR (eRgbAxZm = RGB.BLUE)),
	//
	((eRgbAxYm = RGB.GREEN) OR (eRgbAxYm = RGB.BLUE)),
	((eRgbAxYm = RGB.RED) OR (eRgbAxYm = RGB.BLUE)));
	
	
abyOutData1[7] := usBrightness;
END_METHOD

END_FUNCTION_BLOCK

// xLH_base/app/FB_SDO_READ_4_BYTE
FUNCTION_BLOCK FB_SDO_READ_4_BYTE
VAR_INPUT
	bEnable: BOOL;
	usCoDeviceId: USINT;
	usNetId: USINT := 0;
	uiIndex: UINT;
	usSubindex: USINT;
END_VAR
VAR_OUTPUT
	bDone: BOOL;
	bError: BOOL;
	diValue: DINT;
	udiValue: UDINT;
END_VAR
VAR
	dwAbortCode : DWORD; //contains abort code in case of error
	fbSdoRead4Byte: CIA405.SDO_READ4;	
	fbRtEnable: R_TRIG;
END_VAR

fbRtEnable(CLK:=bEnable);
IF fbRtEnable.CLK THEN
	//bEnable := FALSE;
	bDone := FALSE;
	bError := FALSE;
END_IF

IF fbSdoRead4Byte.CONFIRM THEN
	//value was read without error
	// ==> Copy data from SDO read function block
	MEMUtils.MemCpy(pbyDest := ADR(diValue), pbySrc := ADR(fbSdoRead4Byte.DATA[1]), dwSize := SIZEOF(diValue));
	MEMUtils.MemCpy(pbyDest := ADR(udiValue), pbySrc := ADR(fbSdoRead4Byte.DATA[1]), dwSize := SIZEOF(udiValue));
	//==> On big endian systems: dwValue has to be swapped to CANopen byte order (= Little Endian).
	//MEMUtils.SwapLocalToIntel(pAddress := ADR(diValue), iSize := TO_INT(SIZEOF(diValue))); //function only swaps on big endian systems
	//MEMUtils.SwapLocalToIntel(pAddress := ADR(udiValue), iSize := TO_INT(SIZEOF(udiValue))); //function only swaps on big endian systems
	bDone := TRUE;
	bError := FALSE;
ELSIF fbSdoRead4Byte.ERROR <> CiA405.CANOPEN_KERNEL_ERROR.CANOPEN_KERNEL_NO_ERROR THEN
	//Error occured
	IF fbSdoRead4Byte.ERROR = CIA405.CANOPEN_KERNEL_ERROR.CANOPEN_KERNEL_OTHER_ERROR THEN
		//output error info contains abort code in little endian format
		MEMUtils.MemCpy(pbyDest := ADR(dwAbortCode), pbySrc := ADR(fbSdoRead4Byte.ERRORINFO), dwSize := SIZEOF(dwAbortCode));
		MEMUtils.SwapLocalToIntel(pAddress := ADR(dwAbortCode), iSize := TO_INT(SIZEOF(dwAbortCode))); //function only swaps on big endian systems	
	END_IF
	bDone := FALSE;
	bError := TRUE;
END_IF

fbSdoRead4Byte(
	NETWORK:= CANbus.NetId + 1, //CODESYS NetId starts by 0 (the number entered into the CANbus configurator); CiA405 NETWORK by 1; That is the reason why we have to increment it here.
	ENABLE:= fbRtEnable.CLK,
	TIMEOUT:= 0, //Timeout for SDO read in ms. Here: 0 ==> no timeout
	DEVICE:= usCoDeviceId, // NodeID of destination device
	CHANNEL:= 0, //SDO channel which should be used. 0 means auto channeling ==> the next free channel will be used. It depends on the slave which settings are working here but 0 and channel 1 is always working. 
	INDEX:= uiIndex, //object index which should be read
	SUBINDEX:= usSubindex //object sub index which should be read
);

END_FUNCTION_BLOCK

// xLH_base/app/Visualization
VISUALIZATION Visualization  // 2x2
END_VISUALIZATION
